DATA_BLOCK "ST10Cylinder"
VAR
  Cy : Array[1..110] of "Cyl";
END_VAR
BEGIN
END_DATA_BLOCK
